(*
	Log Warning message to TwinCAT console
*)
{attribute 'hide_all_locals'}
FUNCTION F_LogWarning : BOOL
VAR_INPUT
	sMessage : T_MAXSTRING;
END_VAR

VAR CONSTANT	
	LOGHEADER		: T_MAXSTRING := 'Open Commissioning: %s';
END_VAR

ADSLOGSTR(ADSLOG_MSGTYPE_WARN, LOGHEADER, sMessage);

END_FUNCTION

(* stored: Version 1.1.0.1, ProductVersion 3.1.4024.12
   POU F_LogWarning: Id {0eec24d1-c9c3-06ad-2170-adaf247092ad}, SpecialFunc None *)
